TYPE DUT_MotionStage_Extras :
STRUCT
    fVisuStep: LREAL;
    bVisuLowLim: BOOL;
    bVisuHighLim: BOOL;
END_STRUCT
END_TYPE

(* stored: Version 1.1.0.1, ProductVersion 3.1.4022.18
   DUT DUT_MotionStage_Extras: Id {3e52961b-1e8a-496a-b6ec-5874edc617a6} *)
